// TIA Portal V20 export
DATA_BLOCK "EeMonitor"   // DB61
TITLE = EeMonitor
AUTHOR : SICAR
FAMILY : DB
// Globale EEM Informationen / Global EEM Information
// stored: InstanceOfName LSicar_typeEemDataHmi, InstanceOfType UDT
"LSicar_typeEemDataHmi"
   // VAR
   //    measurePointIndex : USInt := 0;
   //    measConfiguration { ExternalWritable := 'False'} : EnS_EEm_typeMeasConfig;
   //    measOperationHmi { ExternalWritable := 'False'} : EnS_EEm_typeMeasOperation;
   //    work { ExternalWritable := 'False'} : "LSicar_typeEnMeterWorkHmi";
   // END_VAR
BEGIN
   measConfiguration."name" := 'AIEnergyMeter480VACST_EM01';
   measConfiguration.nameShort := 'EM01';
   measConfiguration.media := 'electrical';
   measConfiguration.unitCounterNumber := 1;
   measConfiguration.unitCounterText := 'Wh';
   measConfiguration.unitActValueNumber := 0;
   measConfiguration.unitActValueText := 'W';
   measConfiguration.inputType := 1;
   measConfiguration.type1Counter.overflowCntValue := 1000000.0;
   measConfiguration.type1Counter.normFactor := 1.0;
   measConfiguration.type2ActValue.rawLow := 0.0;
   measConfiguration.type2ActValue.rawHigh := 100.0;
   measConfiguration.type2ActValue.outLow := 0.0;
   measConfiguration.type2ActValue.outHigh := 100.0;
   measOperationHmi.in.counterValue := 277.384918212891;
   measOperationHmi.in.actValue := 0.0;
   measOperationHmi.out.avgValue[0..8] := 0.0;
   measOperationHmi.out.refValue[0..8] := 0.0;
   measOperationHmi.out.differencePercent[0..8] := 0.0;
   measOperationHmi.out.energyCounter[0] := 4.5557861328125;
   measOperationHmi.out.energyCounter[1..8] := 0.0;
   measOperationHmi.out.energyCounterTotal := 4.5557861328125;
   measOperationHmi.out.error := FALSE;
   measOperationHmi.out.energyPerItem := 0.0;
   measOperationHmi.stat.counterLast := 277.473693847656;
   measOperationHmi.stat.counterDifference := 277.384918212891;
   measOperationHmi.stat.startEnergyValue[0..8] := 0.0;
   measOperationHmi.stat.energyCounterIntermediate := 0.0;
   measOperationHmi.stat.energyEnPiCalc[0] := 4.555786;
   measOperationHmi.stat.energyEnPiCalc[1..8] := 0.0;
   work.cycleCounterAvgCalcTod := TOD#00:00:00;
   work.cycleCounterAvgCalcDtl := DTL#1970-01-01-00:00:00;
   work.timePeriodAvgValTod := TOD#00:00:00;
   work.timePeriodAvgValDtl := DTL#1970-01-01-00:00:00;
   work.timePeriodAvgRefTod := TOD#00:00:00;
   work.timePeriodAvgRefDtl := DTL#1970-01-01-00:00:00;
   work.startTimeAvgValLocTime := DTL#1970-01-01-00:00:00;
   work.startTimeAvgRefLocTime := DTL#1970-01-01-00:00:00;
   work.numberOfRecords := 209;
END_DATA_BLOCK
